// TIA Portal V18 export
TYPE "UDT_sirene"
// stored: IsFailsafeCompliant false
   STRUCT
      toneSelect { ExternalVisible := 'False'; S7_SetPoint := 'True'} : Int;
      toneDuration { ExternalVisible := 'False'; S7_SetPoint := 'True'} : Time;
      trigger { ExternalVisible := 'False'} : Bool;
      test { ExternalVisible := 'False'} : Bool;
   END_STRUCT;
END_TYPE
